(* CODESYS project TcUnit.library
   Company: TcUnit
   DefaultNamespace: TcUnit
   Version: 0.0.0.2
   Placeholder: TcUnit
   Title: TcUnit

Project tree, tasks and I/O mapping:
  libraries: Tc2_Standard, * (Beckhoff Automation GmbH); Tc2_System, * (Beckhoff Automation GmbH); Tc2_Utilities, * (Beckhoff Automation GmbH); Tc3_Interfaces, * (Beckhoff Automation GmbH); Tc3_Module, * (Beckhoff Automation GmbH)
  DUTs/
  GVLs/
  POUs/
    function block FB_Assert [ST]: AbortAfterFail, AreEqualBOOL, AreEqualBYTE, AreEqualDINT, AreEqualDWORD, AreEqualGUID, AreEqualHRESULT, AreEqualINT, AreEqualLINT, AreEqualLREAL, AreEqualLTIME, AreEqualLWORD, AreEqualMEM, AreEqualREAL, AreEqualSINT, AreEqualSTRING, AreEqualTIME, AreEqualUDINT, AreEqualUINT, AreEqualULINT, AreEqualUSINT, AreEqualWORD, FB_init, IsFalse, IsTrue, MultipleLog, PrintFailed, PrintPassed, State, StateMachineError
  Version/
    global variables Global_Version
  00000000-0000-0000-0000-000000000000|TcUnit.tmc
  TcUnit.tmc
*)

// Version/Global_Version
{attribute 'TcGenerated'}
// This function has been automatically generated from the project information.
VAR_GLOBAL CONSTANT
	{attribute 'const_non_replaced'}
	{attribute 'linkalways'}
	stLibVersion_TcUnit : ST_LibVersion := (iMajor := 0, iMinor := 0, iBuild := 0, iRevision := 2, sVersion := '0.0.0.2');
END_VAR

// POUs/FB_Assert
FUNCTION_BLOCK PUBLIC FB_Assert
VAR
	bMultipleLogFlag	: BOOL;
	bAbortAfterFailFlag	: BOOL;
	bAbort				: BOOL;
	nState				: UDINT;
	sInstanceName		: STRING[255];
	sLastInstance		: STRING[255];
	sLastMessage		: STRING[255];
	nLastState			: UDINT;
END_VAR

{attribute 'monitoring':='call'}
PROPERTY PUBLIC AbortAfterFail : BOOL
SET
THIS^.bAbortAfterFailFlag := AbortAfterFail;
END_SET
END_PROPERTY

METHOD PUBLIC AreEqualBOOL : BOOL
VAR_INPUT
	bExpected	: BOOL;
	bActual		: BOOL;
	sMessage	: STRING(80);
END_VAR
IF (bExpected <> bActual) THEN
	PrintFailed(TO_STRING(bActual), TO_STRING(bExpected), '', sMessage, 'BOOL');
	AreEqualBOOL := FALSE;
ELSE
	AreEqualBOOL := TRUE;
END_IF
END_METHOD

METHOD PUBLIC AreEqualBYTE : BOOL
VAR_INPUT
	nExpected	: BYTE;
	nActual		: BYTE;
	sMessage	: STRING(80);
END_VAR
IF (nExpected <> nActual) THEN
	PrintFailed(CONCAT('16#', DWORD_TO_HEXSTR(TO_DWORD(nActual), 8, FALSE)),
				CONCAT('16#', DWORD_TO_HEXSTR(TO_DWORD(nExpected), 8, FALSE)),
				'',
				sMessage,
				'BYTE');
	AreEqualBYTE := FALSE;
ELSE
	AreEqualBYTE := TRUE;
END_IF
END_METHOD

METHOD PUBLIC AreEqualDINT : BOOL
VAR_INPUT
	nExpected	: DINT;
	nActual		: DINT;
	sMessage	: STRING(80);
END_VAR
IF (nExpected <> nActual) THEN
	PrintFailed(TO_STRING(nActual), TO_STRING(nExpected), '', sMessage, 'DINT');
	AreEqualDINT := FALSE;
ELSE
	AreEqualDINT := TRUE;
END_IF
END_METHOD

METHOD PUBLIC AreEqualDWORD : BOOL
VAR_INPUT
	nExpected	: DWORD;
	nActual		: DWORD;
	sMessage	: STRING(80);
END_VAR
IF (nExpected <> nActual) THEN
	PrintFailed(CONCAT('16#', DWORD_TO_HEXSTR(nActual, 8, FALSE)),
				CONCAT('16#', DWORD_TO_HEXSTR(nExpected, 8, FALSE)),
				'',
				sMessage,
				'DWORD');
	AreEqualDWORD := FALSE;
ELSE
	AreEqualDWORD := TRUE;
END_IF
END_METHOD

METHOD PUBLIC AreEqualGUID : BOOL
VAR_INPUT
	stExpected	: GUID;
	stActual	: GUID;
	sMessage	: STRING(80);
END_VAR
VAR
	nIdx		: BYTE;
	bEqual		: BOOL;
END_VAR
bEqual := TRUE;
bEqual := bEqual AND stExpected.Data1 = stActual.Data1;
bEqual := bEqual AND stExpected.Data2 = stActual.Data2;
bEqual := bEqual AND stExpected.Data3 = stActual.Data3;

FOR nIdx := 0 TO 7 DO
	bEqual := bEqual AND (stExpected.Data4[nIdx] = stActual.Data4[nIdx]);
END_FOR

IF (NOT bEqual) THEN
	PrintFailed('', '', '', sMessage, 'GUID');
	AreEqualGUID := FALSE;
ELSE
	AreEqualGUID := TRUE;
END_IF
END_METHOD

METHOD PUBLIC AreEqualHRESULT : BOOL
VAR_INPUT
	hResultExp	: hResult;
	hResultAct	: hResult;
	sMessage	: STRING(80);
END_VAR
IF (hResultExp <> hResultAct) THEN
	PrintFailed(CONCAT('16#', DWORD_TO_HEXSTR(TO_DWORD(hResultAct), 8, FALSE)),
				CONCAT('16#', DWORD_TO_HEXSTR(TO_DWORD(hResultExp), 8, FALSE)),
				'',
				sMessage,
				'HRESULT');
	AreEqualHRESULT := FALSE;
ELSE
	AreEqualHRESULT := TRUE;
END_IF
END_METHOD

METHOD PUBLIC AreEqualINT : BOOL
VAR_INPUT
	nExpected	: INT;
	nActual		: INT;
	sMessage	: STRING(80);
END_VAR
IF (nExpected <> nActual) THEN
	PrintFailed(TO_STRING(nActual), TO_STRING(nExpected), '', sMessage, 'INT');
	AreEqualINT := FALSE;
ELSE
	AreEqualINT := TRUE;
END_IF
END_METHOD

METHOD PUBLIC AreEqualLINT : BOOL
VAR_INPUT
	nExpected	: LINT;
	nActual		: LINT;
	sMessage	: STRING(80);
END_VAR
IF (nExpected <> nActual) THEN
	PrintFailed(TO_STRING(nActual), TO_STRING(nExpected), '', sMessage, 'LINT');
	AreEqualLINT := FALSE;
ELSE
	AreEqualLINT := TRUE;
END_IF
END_METHOD

METHOD PUBLIC AreEqualLREAL : BOOL
VAR_INPUT
	fExpected	: LREAL;
	fActual		: LREAL;
	fTolerance	: LREAL;
	sMessage	: STRING(80);
END_VAR
VAR
	fbFormatActual		: FB_FormatString;
	fbFormatExpected	: FB_FormatString;
	sFormatOption		: STRING(20);
END_VAR
IF (ABS(fExpected-fActual) > fTolerance) THEN
	IF (fTolerance >= 0.1) THEN
		sFormatOption := '%4.1F';
	ELSIF (fTolerance >= 0.01) THEN
		sFormatOption := '%4.2F';
	ELSIF (fTolerance >= 0.001) THEN
		sFormatOption := '%4.3F';
	ELSIF (fTolerance >= 0.000001) THEN
		sFormatOption := '%4.6F';
	ELSE
		sFormatOption := '%4.9F';
	END_IF

	fbFormatActual(sFormat := sFormatOption, arg1 := F_LREAL(fActual));
	fbFormatExpected(sFormat := sFormatOption, arg1 := F_LREAL(fExpected));

	PrintFailed(fbFormatActual.sOut, fbFormatExpected.sOut, TO_STRING(fTolerance), sMessage, 'LREAL');
	AreEqualLREAL := FALSE;
ELSE
	AreEqualLREAL := TRUE;
END_IF
END_METHOD

METHOD PUBLIC AreEqualLTIME : BOOL
VAR_INPUT
	tExpected		: LTIME;
	tActual			: LTIME;
	tTolerance		: LTIME;
	sMessage		: STRING(80);
END_VAR
IF (tActual < (tExpected - tTolerance)) OR (tActual > (tExpected + tTolerance)) THEN
	PrintFailed(TO_STRING(tActual), TO_STRING(tExpected), TO_STRING(tTolerance), sMessage, 'LTIME');
	AreEqualLTIME := FALSE;
ELSE
	AreEqualLTIME := TRUE;
END_IF
END_METHOD

METHOD PUBLIC AreEqualLWORD : BOOL
VAR_INPUT
	nExpected	: LWORD;
	nActual		: LWORD;
	sMessage	: STRING(80);
END_VAR
IF (nExpected <> nActual) THEN
	PrintFailed(CONCAT('16#', LWORD_TO_HEXSTR(nActual, 16, FALSE)),
				CONCAT('16#', LWORD_TO_HEXSTR(nExpected, 16, FALSE)),
				'',
				sMessage,
				'LWORD');
	AreEqualLWORD := FALSE;
ELSE
	AreEqualLWORD := TRUE;
END_IF
END_METHOD

METHOD PUBLIC AreEqualMEM : BOOL
VAR_INPUT
	pExpected	: PVOID;
	pActual		: PVOID;
	nSize		: UDINT;
	sMessage	: STRING(80);
END_VAR
IF (MEMCMP(pExpected, pActual, nSize) <> 0) THEN
	PrintFailed('', '', '', sMessage, 'MEM');
	AreEqualMEM := FALSE;
ELSE
	AreEqualMEM := TRUE;
END_IF
END_METHOD

METHOD PUBLIC AreEqualREAL : BOOL
VAR_INPUT
	fExpected	: REAL;
	fActual		: REAL;
	fTolerance	: REAL;
	sMessage	: STRING(80);
END_VAR
VAR
	fbFormatActual		: FB_FormatString;
	fbFormatExpected	: FB_FormatString;
	sFormatOption		: STRING(20);
END_VAR
IF (ABS(fExpected-fActual) > fTolerance) THEN
	IF (fTolerance >= 0.1) THEN
		sFormatOption := '%4.1F';
	ELSIF (fTolerance >= 0.01) THEN
		sFormatOption := '%4.2F';
	ELSIF (fTolerance >= 0.001) THEN
		sFormatOption := '%4.3F';
	ELSIF (fTolerance >= 0.000001) THEN
		sFormatOption := '%4.6F';
	ELSE
		sFormatOption := '%4.9F';
	END_IF

	fbFormatActual(sFormat := sFormatOption, arg1 := F_Real(fActual));
	fbFormatExpected(sFormat := sFormatOption, arg1 := F_Real(fExpected));

	PrintFailed(fbFormatActual.sOut, fbFormatExpected.sOut, TO_STRING(fTolerance), sMessage, 'REAL');
	AreEqualREAL := FALSE;
ELSE
	AreEqualREAL := TRUE;
END_IF
END_METHOD

METHOD PUBLIC AreEqualSINT : BOOL
VAR_INPUT
	nExpected	: SINT;
	nActual		: SINT;
	sMessage	: STRING(80);
END_VAR
IF (nExpected <> nActual) THEN
	PrintFailed(TO_STRING(nActual), TO_STRING(nExpected), '', sMessage, 'SINT');
	AreEqualSINT := FALSE;
ELSE
	AreEqualSINT := TRUE;
END_IF
END_METHOD

METHOD PUBLIC AreEqualSTRING : BOOL
VAR_INPUT
	sExpected	: STRING(255);
	sActual		: STRING(255);
	sMessage	: STRING(80);
END_VAR
IF (sExpected <> sActual) THEN
	PrintFailed(sActual, sExpected, '', sMessage, 'STRING');
	AreEqualSTRING := FALSE;
ELSE
	AreEqualSTRING := TRUE;
END_IF
END_METHOD

METHOD PUBLIC AreEqualTIME : BOOL
VAR_INPUT
	tExpected		: TIME;
	tActual			: TIME;
	tTolerance		: TIME;
	sMessage		: STRING(80);
END_VAR
IF (tActual < (tExpected - tTolerance)) OR (tActual > (tExpected + tTolerance)) THEN
	PrintFailed(TO_STRING(tActual), TO_STRING(tExpected), TO_STRING(tTolerance), sMessage, 'TIME');
	AreEqualTIME := FALSE;
ELSE
	AreEqualTIME := TRUE;
END_IF
END_METHOD

METHOD PUBLIC AreEqualUDINT : BOOL
VAR_INPUT
	nExpected	: UDINT;
	nActual		: UDINT;
	sMessage	: STRING(80);
END_VAR
IF (nExpected <> nActual) THEN
	PrintFailed(TO_STRING(nActual), TO_STRING(nExpected), '', sMessage, 'UDINT');
	AreEqualUDINT := FALSE;
ELSE
	AreEqualUDINT := TRUE;
END_IF
END_METHOD

METHOD PUBLIC AreEqualUINT : BOOL
VAR_INPUT
	nExpected	: UINT;
	nActual		: UINT;
	sMessage	: STRING(80);
END_VAR
IF (nExpected <> nActual) THEN
	PrintFailed(TO_STRING(nActual), TO_STRING(nExpected), '', sMessage, 'UINT');
	AreEqualUINT := FALSE;
ELSE
	AreEqualUINT := TRUE;
END_IF
END_METHOD

METHOD PUBLIC AreEqualULINT : BOOL
VAR_INPUT
	nExpected	: ULINT;
	nActual		: ULINT;
	sMessage	: STRING(80);
END_VAR
IF (nExpected <> nActual) THEN
	PrintFailed(TO_STRING(nActual), TO_STRING(nExpected), '', sMessage, 'ULINT');
	AreEqualULINT := FALSE;
ELSE
	AreEqualULINT := TRUE;
END_IF
END_METHOD

METHOD PUBLIC AreEqualUSINT : BOOL
VAR_INPUT
	nExpected	: USINT;
	nActual		: USINT;
	sMessage	: STRING(80);
END_VAR
IF (nExpected <> nActual) THEN
	PrintFailed(TO_STRING(nActual), TO_STRING(nExpected), '', sMessage, 'USINT');
	AreEqualUSINT := FALSE;
ELSE
	AreEqualUSINT := TRUE;
END_IF
END_METHOD

METHOD PUBLIC AreEqualWORD : BOOL
VAR_INPUT
	nExpected	: WORD;
	nActual		: WORD;
	sMessage	: STRING(80);
END_VAR
IF (nExpected <> nActual) THEN
	PrintFailed(CONCAT('16#', DWORD_TO_HEXSTR(TO_DWORD(nActual), 8, FALSE)),
				CONCAT('16#', DWORD_TO_HEXSTR(TO_DWORD(nExpected), 8, FALSE)),
				'',
				sMessage,
				'WORD');
	AreEqualWORD := FALSE;
ELSE
	AreEqualWORD := TRUE;
END_IF
END_METHOD

METHOD FB_init : BOOL
VAR_INPUT
	bInitRetains : BOOL; // if TRUE, the retain variables are initialized (warm start / cold start)
	bInCopyCode : BOOL;  // if TRUE, the instance afterwards gets moved into the copy code (online change)
	sInstanceName : STRING(255);
END_VAR
THIS^.sInstanceName := sInstanceName;
END_METHOD

METHOD PUBLIC IsFalse : BOOL
VAR_INPUT
	bCondition	: BOOL;
	sMessage	: STRING(80);
END_VAR
IF bCondition THEN
	PrintFailed(BOOL_TO_STRING(bCondition), 'FALSE', '', sMessage, 'BOOL');
	IsFalse := FALSE;
ELSE
	IsFalse := TRUE;
END_IF
END_METHOD

METHOD PUBLIC IsTrue : BOOL
VAR_INPUT
	bCondition	: BOOL;
	sMessage	: STRING(80);
END_VAR
IF (NOT bCondition) THEN
	PrintFailed(TO_STRING(bCondition), 'TRUE', '', sMessage, 'BOOL');
	IsTrue := FALSE;
ELSE
	IsTrue := TRUE;
END_IF
END_METHOD

{attribute 'monitoring':='call'}
PROPERTY PUBLIC MultipleLog : BOOL
SET
THIS^.bMultipleLogFlag := MultipleLog;
END_SET
END_PROPERTY

METHOD PUBLIC PrintFailed
VAR_INPUT
	sActual		: STRING(80);
	sExpected	: STRING(80);
	sTolerance	: STRING(80);
	sMessage	: STRING(80);
	sType		: STRING(20);
END_VAR
VAR
	sState		: STRING(10);
	sString		: STRING(255);
END_VAR
IF ((THIS^.sLastMessage <> sMessage) OR (THIS^.nLastState <> THIS^.nState) OR THIS^.bMultipleLogFlag) THEN
	THIS^.sLastInstance := THIS^.sInstanceName;
	THIS^.sLastMessage := sMessage;
	THIS^.nLastState := THIS^.nState;
	
	sString := THIS^.sInstanceName;

	sState := DWORD_TO_HEXSTR(TO_DWORD(THIS^.nState), 4, FALSE);
	
	sString := CONCAT(sString, '; State: 16#');
	sString := CONCAT(sString, sState);
	
	IF (LEN(sType) > 0) THEN
		sString := CONCAT(sString, '; ');
		sString := CONCAT(sString, sType);
	END_IF
	
	IF (LEN(sMessage) > 0) THEN
		sString := CONCAT(sString, '; ');
		sString := CONCAT(sString, sMessage);
	END_IF
	
	IF (LEN(sActual) > 0) THEN
		sString := CONCAT(sString, '; Act: ');
		sString := CONCAT(sString, sActual);
	END_IF
	
	IF (LEN(sExpected) > 0) THEN
		sString := CONCAT(sString, '; Exp: ');
		sString := CONCAT(sString, sExpected);
	END_IF
	
	IF (LEN(sTolerance) > 0) THEN
		sString := CONCAT(sString, '; Tol: ');
		sString := CONCAT(sString, sTolerance);
	END_IF
	
	ADSLOGSTR(msgCtrlMask := ADSLOG_MSGTYPE_ERROR, msgFmtStr := 'Failed: %s', strArg := sString);					
				
	IF (THIS^.bAbortAfterFailFlag) THEN
		THIS^.bAbort := TRUE;
	END_IF
END_IF
END_METHOD

METHOD PUBLIC PrintPassed
VAR_INPUT
	sMessage	: STRING(80);
END_VAR
VAR
	sState		: STRING(10);
	sString		: STRING(255);	
END_VAR
IF ((THIS^.sLastMessage <> sMessage) OR (THIS^.nLastState <> THIS^.nState) OR THIS^.bMultipleLogFlag) THEN
	THIS^.sLastInstance := THIS^.sInstanceName;
	THIS^.sLastMessage := sMessage;
	THIS^.nLastState := THIS^.nState;
	
	sString := THIS^.sInstanceName;

	sState := DWORD_TO_HEXSTR(TO_DWORD(THIS^.nState), 4, FALSE);
	
	sString := CONCAT(sString, '; State: 16#');
	sString := CONCAT(sString, sState);
		
	IF (LEN(sMessage) > 0) THEN
		sString := CONCAT(sString, '; ');
		sString := CONCAT(sString, sMessage);
	END_IF
		
	ADSLOGSTR(msgCtrlMask := ADSLOG_MSGTYPE_WARN, msgFmtStr := 'Passed: %s', strArg := sString);
END_IF
END_METHOD

PROPERTY PUBLIC State : UDINT
GET
State := THIS^.nState;
END_GET
SET
IF (THIS^.bAbort) THEN
	THIS^.nState := 16#FFFF;
ELSE
	THIS^.nState := LIMIT(0, State, 16#FFFF);
END_IF
END_SET
END_PROPERTY

METHOD PUBLIC StateMachineError : BOOL
PrintFailed('', '', '', 'Invalid State!', 'StateMachine');
THIS^.nState := 16#FFFF;
END_METHOD

END_FUNCTION_BLOCK
